ABB RobotStudio station: burguerBot.rsstn

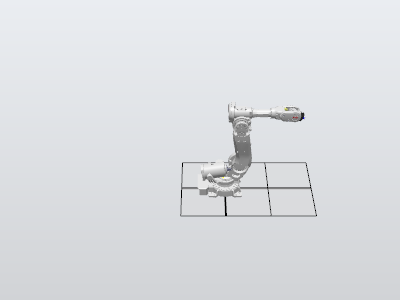
Station Station (saved by RobotStudio 24.1.10713.1)
Controller IRB140_6_81_1
  mechanical unit ROB_1: ?, 6 joints, base frame (0, 0, 0) mm
Layout (positions relative to the parent item):
  - IRB6640_180_255__04 [mechanism, from %ABB.RobotStudio.Models.IRB6640%\IRB6640_180_255_G_04.rslib] at (0, 0, 0) mm; joint values [0, 0, 0, 0, 0.5236, 0] (rad or m)
